Yaskawa INFORM job: SVETS2.JBI

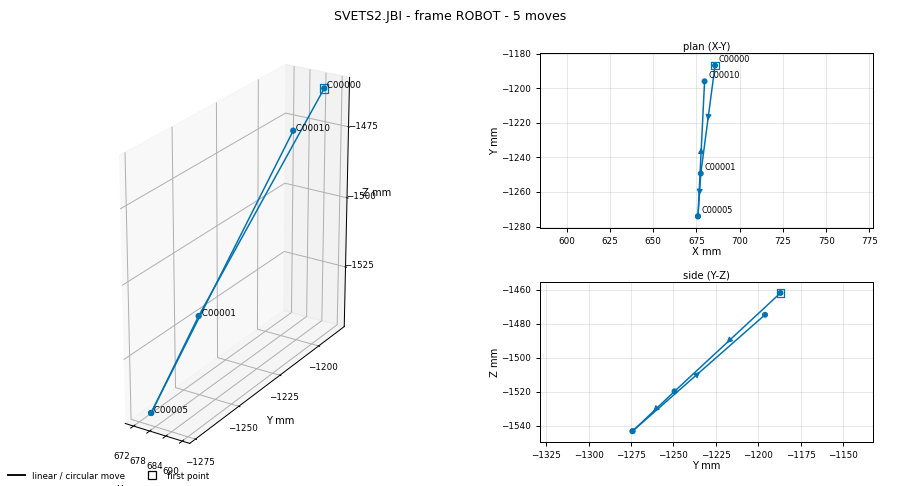
[picture p0: tool path of SVETS2.JBI in frame ROBOT, 5 of 5 moves have a stored position in this frame; points joined in program order, loops and branches not executed]
/JOB
//NAME SVETS2
///FOLDERNAME FOLDER001
//POS
///NPOS 11,11,0,0,0,0
///TOOL 0
///POSTYPE ROBOT
///RECTAN
///RCONF 0,0,0,0,0,0,0,0,0,0,0,0,0,0,0,0,0,0,0,0,0,0,0,0
C00000=685.754,-1186.880,-1461.862,-47.3471,1.8058,-5.8615
C00001=677.505,-1249.321,-1519.831,-47.3472,1.8056,-5.8618
C00002=677.505,-1249.321,-1519.831,-47.3472,1.8056,-5.8618
C00003=677.510,-1261.615,-1519.826,-47.3467,1.8037,-5.8631
C00004=677.504,-1249.321,-1531.924,-47.3469,1.8046,-5.8627
///RCONF 0,0,0,0,1,0,0,0,0,0,0,0,0,0,0,0,0,0,0,0,0,0,0,0
C00005=675.869,-1274.090,-1543.336,-47.3473,1.8088,-5.8618
///RCONF 0,0,0,0,0,0,0,0,0,0,0,0,0,0,0,0,0,0,0,0,0,0,0,0
C00006=675.912,-1261.479,-1484.682,-47.3483,1.8046,-5.8620
C00007=675.894,-1215.863,-1531.107,-47.3476,1.8067,-5.8614
C00008=670.755,-1263.692,-1537.553,-47.3480,1.8066,-5.8620
///RCONF 0,0,0,0,1,0,0,0,0,0,0,0,0,0,0,0,0,0,0,0,0,0,0,0
C00009=675.869,-1274.090,-1543.336,-47.3473,1.8088,-5.8618
///RCONF 0,0,0,0,0,0,0,0,0,0,0,0,0,0,0,0,0,0,0,0,0,0,0,0
C00010=679.698,-1195.993,-1474.712,-47.3474,1.8066,-5.8623
BC00000=539.753,2775.784,452.161
BC00001=539.753,2775.784,452.161
BC00002=539.753,2775.784,452.161
BC00003=539.753,2775.784,452.161
BC00004=539.753,2775.784,452.161
BC00005=539.753,2775.784,452.161
BC00006=539.753,2775.784,452.161
BC00007=539.753,2775.784,452.161
BC00008=789.919,2775.784,452.161
BC00009=768.617,2783.205,452.161
BC00010=789.919,2775.784,452.161
//INST
///DATE 2023/07/12 09:41
///ATTR SC,RW,RJ
////FRAME ROBOT
///GROUP1 RB1,BS1
NOP
MOVL C00000 BC00000 V=150.0
MACRO1 MJ#(0) ARGF4
MOVL C00001 BC00001 V=75.0
REFP 4 C00002 BC00002
REFP 5 C00003 BC00003
REFP 6 C00004 BC00004
MOVL C00005 BC00005 V=75.0
REFP 1 C00006 BC00006
REFP 2 C00007 BC00007
REFP 3 C00008 BC00008
ARCON
WVON WEV#(1)
MOVL C00009 BC00009 V=7.5
WVOF
ARCOF
SFTOF
MOVL C00010 BC00010 V=150.0
END
